// TIA Portal V19 export
TYPE "LEXCHANGETRAY_typeConstraintRollerEm_toConstraintWorkstationDeliver"
// stored: Access Published
   STRUCT
      feedback : "LEXCHANGETRAY_typeConstraintRollerEm_toConstraintWorkstationFeedback";
      req : "LEXCHANGETRAY_typeConstraintRollerEm_toConstraintWorkstationReq";
   END_STRUCT;
END_TYPE
